FUNCTION_BLOCK EL7201
VAR_INPUT
END_VAR
VAR_OUTPUT
END_VAR
VAR
END_VAR

END_FUNCTION_BLOCK

(* stored: Version 1.1.0.1, ProductVersion 3.1.4022.17
   POU EL7201: Id {41c27df6-567d-42f4-a342-26c06a4b0130}, SpecialFunc None *)
